(* PLC project TestProject, Test Test 1.0 *)
(* stored: creationDateTime 2024-01-01T00:00:00 *)

FUNCTION_BLOCK Counter
  VAR_INPUT
    Reset : BOOL;
  END_VAR
  VAR_OUTPUT
    Count : INT;
  END_VAR

            IF Reset THEN
  Count := 0;
END_IF;
          
END_FUNCTION_BLOCK

PROGRAM Main
  VAR
    MyCounter : Counter;
  END_VAR

            MyCounter(Reset := FALSE);
          
END_PROGRAM
